Fanuc KAREL source: kd00016.KL

PROGRAM KD00016
%NOLOCKGROUP
VAR
I:INTEGER;J:INTEGER;B:BOOLEAN;R:REAL;S : STRING[80]
BEGIN
--
--
--
--
I=0
CONNECT TIMER TO I
END KD00016
